// TIA Portal V19 export
TYPE "type_xyzRequestData"
// stored: Access Published, Namespace Unit3
   STRUCT
      xyzEnabled : Bool;   // 允许运动
   END_STRUCT;
END_TYPE
